FUNCTION_BLOCK RT_E_PERMIT (* Permissive propagation of an event *)
  (* Standard: 61499-1-A.1 *)
  (* Version 0.0, 2008-07-10, 4DIAC-IDE, 4DIAC-Consortium *)
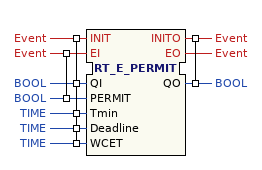
  EVENT_INPUT
    INIT WITH QI, Tmin, Deadline, WCET;
    EI WITH PERMIT; (* Event input *)
  END_EVENT
  EVENT_OUTPUT
    INITO WITH QO;
    EO; (* Event output *)
  END_EVENT
  VAR_INPUT
    QI : BOOL;
    PERMIT : BOOL;
    Tmin : TIME;
    Deadline : TIME;
    WCET : TIME;
  END_VAR
  VAR_OUTPUT
    QO : BOOL;
  END_VAR
END_FUNCTION_BLOCK
